// Mitsubishi GX Works2 project: setak   PLC: Q03UDV

PROGRAM MAIN
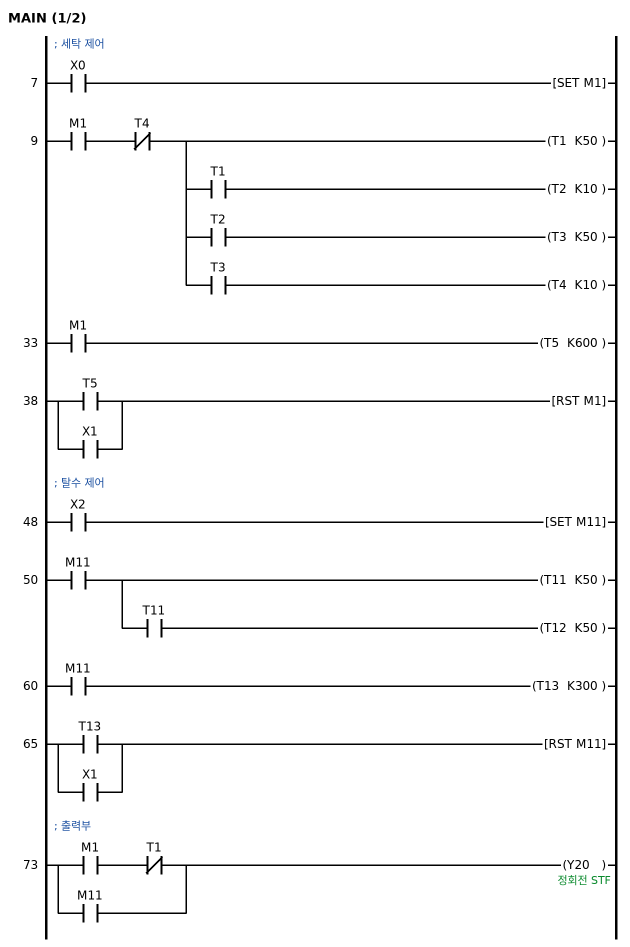
; 세탁 제어
7     LD      X0
      SET     M1
9     LD      M1
      ANI     T4
      OUT     T1 K50
      MPS
      AND     T1
      OUT     T2 K10
      MRD
      AND     T2
      OUT     T3 K50
      MPP
      AND     T3
      OUT     T4 K10
33    LD      M1
      OUT     T5 K600
38    LD      T5
      OR      X1
      RST     M1
; 탈수 제어
48    LD      X2
      SET     M11
50    LD      M11
      OUT     T11 K50
      AND     T11
      OUT     T12 K50
60    LD      M11
      OUT     T13 K300
65    LD      T13
      OR      X1
      RST     M11
; 출력부
73    LD      M1
      ANI     T1
      OR      M11
      OUT     Y20  ; 정회전 STF
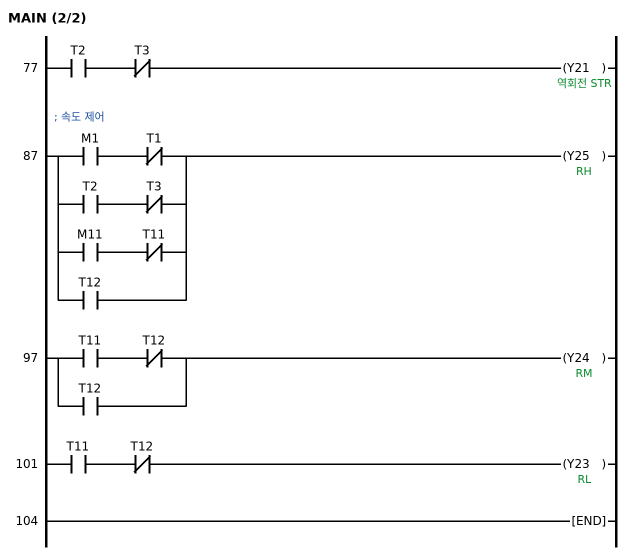
77    LD      T2
      ANI     T3
      OUT     Y21  ; 역회전 STR
; 속도 제어
87    LD      M1
      ANI     T1
      LD      T2
      ANI     T3
      ORB
      LD      M11
      ANI     T11
      ORB
      OR      T12
      OUT     Y25  ; RH
97    LD      T11
      ANI     T12
      OR      T12
      OUT     Y24  ; RM
101   LD      T11
      ANI     T12
      OUT     Y23  ; RL
104   END
END_PROGRAM

PROGRAM speedBit
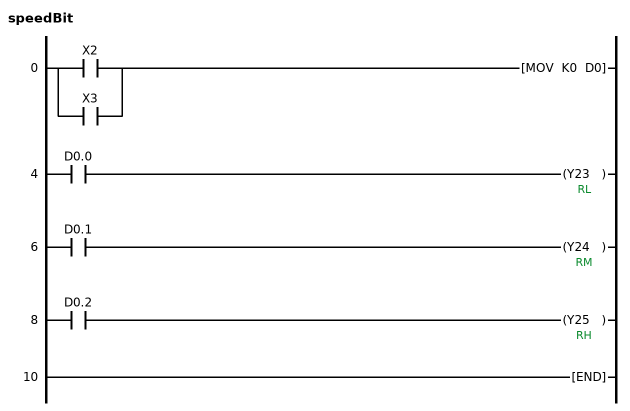
0     LD      X2
      OR      X3
      MOV     K0 D0
4     LD      D0.0
      OUT     Y23  ; RL
6     LD      D0.1
      OUT     Y24  ; RM
8     LD      D0.2
      OUT     Y25  ; RH
10    END
END_PROGRAM
